VAR_GLOBAL
END_VAR

(* stored: Version 1.1.0.1, ProductVersion 3.1.0.20
   GVL RFD_Constants: Id {6f1bed1e-6340-4698-9eec-8e2b1ccc5445} *)
